% RSLogix 500 project LVD200607_TestA.RSS, saved by version 11.00.00.00 %
PROJECT "LINL0619"    % processor: type code 64 %

PROGRAM FILES
  LAD 2 "MAIN"  50 rungs  % Main Program Routine %
  LAD 4 "ENABLES"  14 rungs
  LAD 6 "FEED"  11 rungs  % normal %
  LAD 8 "SPEEDS"  12 rungs
  LAD 20 "HSC BOT"  5 rungs
  LAD 22 "HSC TOP"  5 rungs
  LAD 30 "1 MS STI"  17 rungs  % high speed %
  LAD 40 "SHIFT BOT"  8 rungs
  LAD 42 "SHIFT TOP"  16 rungs
  LAD 50 "BOTOPTIC"  3 rungs
  LAD 52 "BOTOPTMES"  7 rungs
  LAD 60 "1 INS1"  23 rungs
  LAD 61 "2 INS1RESU"  7 rungs
  LAD 62 "3 INS1PASS"  5 rungs
  LAD 63 "4 INS1FAIL"  3 rungs
  LAD 64 "5 INS1ACQ"  8 rungs
  LAD 65 "6 Q1TESTTR"  5 rungs
  LAD 66 "7 INS1TRIG"  5 rungs
  LAD 67 "8 FIFO1SET"  9 rungs
  LAD 68 "9 FIFO1GET"  8 rungs
  LAD 69 "10INSDATA1"  3 rungs
  LAD 70 "11TSTFALT1"  9 rungs
  LAD 71 "12INS1FIX1"  5 rungs
  LAD 72 "13INS1FIX2"  3 rungs
  LAD 73 "14 HSTRIG1"  5 rungs
  LAD 80 "XFER"  3 rungs
  LAD 90 "TOPOPTIC"  10 rungs
  LAD 91 "TOPOPVERT"  13 rungs
  LAD 92 "TOPOPREAL"  19 rungs
  LAD 93 "TOPOPTEST"  8 rungs
  LAD 94 "TOPOPRANGE"  6 rungs
  LAD 95 "TOPOPOKAY"  6 rungs
  LAD 96 "TESTINJECT"  8 rungs
  LAD 100 "1 INS5"  23 rungs
  LAD 101 "2 INS5RESU"  7 rungs
  LAD 102 "3 INS5PASS"  5 rungs
  LAD 103 "4 INS5FAIL"  3 rungs
  LAD 104 "5 INS5ACQ"  8 rungs
  LAD 105 "6 Q5TESTTR"  5 rungs
  LAD 106 "7 INS5TRIG"  5 rungs
  LAD 107 "8 FIFO5SET"  9 rungs
  LAD 108 "9 FIFO5GET"  8 rungs
  LAD 109 "10INSDATA5"  3 rungs
  LAD 110 "11TSTFALT5"  9 rungs
  LAD 111 "12INS5FIX1"  5 rungs
  LAD 112 "13INS5FIX2"  3 rungs
  LAD 113 "14 HSTRIG5"  5 rungs
  LAD 120 "1 INS6"  23 rungs
  LAD 121 "2 INS6RESU"  7 rungs
  LAD 122 "3 INS6PASS"  5 rungs
  LAD 123 "4 INS6FAIL"  3 rungs
  LAD 124 "5 INS6ACQ"  8 rungs
  LAD 125 "6 Q6TESTTR"  5 rungs
  LAD 126 "7 INS6TRIG"  5 rungs
  LAD 127 "8 FIFO6SET"  9 rungs
  LAD 128 "9 FIFO6GET"  8 rungs
  LAD 129 "10INSDATA6"  3 rungs
  LAD 130 "11TSTFALT6"  9 rungs
  LAD 131 "12INS6FIX1"  5 rungs
  LAD 132 "13INS6FIX2"  3 rungs
  LAD 133 "14 HSTRIG6"  5 rungs
  LAD 190 "PASS BLOW"  13 rungs
  LAD 201 "UNUSED"  14 rungs
  LAD 215 "TESTTRIG1"  4 rungs
  LAD 216 "TESTTRIG5"  4 rungs
  LAD 217 "TESTTRIG6"  4 rungs
  LAD 219 "PACKAGER"  28 rungs  % normal %
  LAD 220 "NO PACKAGE"  8 rungs
  LAD 222 "RATE1"  9 rungs
  LAD 223 "RATE2"  6 rungs
  LAD 224 "RESET RATE"  6 rungs
  LAD 240 "NP STOP"  8 rungs
  LAD 246 "SPEED BOT"  8 rungs  % high speed %
  LAD 248 "SPEED TOP"  8 rungs  % high speed %
  LAD 250 "P BOT"  7 rungs  % high speed %
  LAD 252 "P TOP"  7 rungs  % high speed %
  LAD 254 "TOTALCOUNT"  4 rungs
  LAD 255 "BLANK"  1 rungs
  LAD 74, 81, 114, 134, 191, 214, 218, 221, 225, 241: only END

DATA FILES
  O0 OUTPUT  11 elements
  I1 INPUT  11 elements
  S2 STATUS  66 elements
  B3 BINARY  14 elements
  T4 TIMER  45 elements
  C5 COUNTER  1 elements
  R6 CONTROL  30 elements
  N7 INTEGER  200 elements
  F8 FLOAT  100 elements
  B12 HMI_BINARY  22 elements  % general use with hmi to avoid additional reads %
  L13  COUNTS  256 elements
  F14 HMI_FLOATS  100 elements
  N15 HMI_INTS  100 elements
  L16 HMI_LONGS  100 elements
  L19 RATE DATA  50 elements
  L28 INS1TIME  50 elements
  L29 INS1POS  50 elements
  L30 INS5TIME  50 elements
  L31 INS5POS  50 elements
  L32 INS6TIME  50 elements
  L33 INS6POS  50 elements
  B34 BOT NG  128 elements
  B35 TOP NG  128 elements
  B36 BOTGOOD  128 elements
  B37 TOPGOOD  128 elements
  B38 EX1 TEST  128 elements
  B39 EX2GOOD  128 elements
  B40 EX2 TEST  128 elements
  N184 TEST INTS  50 elements
  L192 SPD OFFSET  50 elements
  B196 CTRL BITS  50 elements
  L199 USED  36 elements

LADDER 2 "MAIN"    % Main Program Routine %
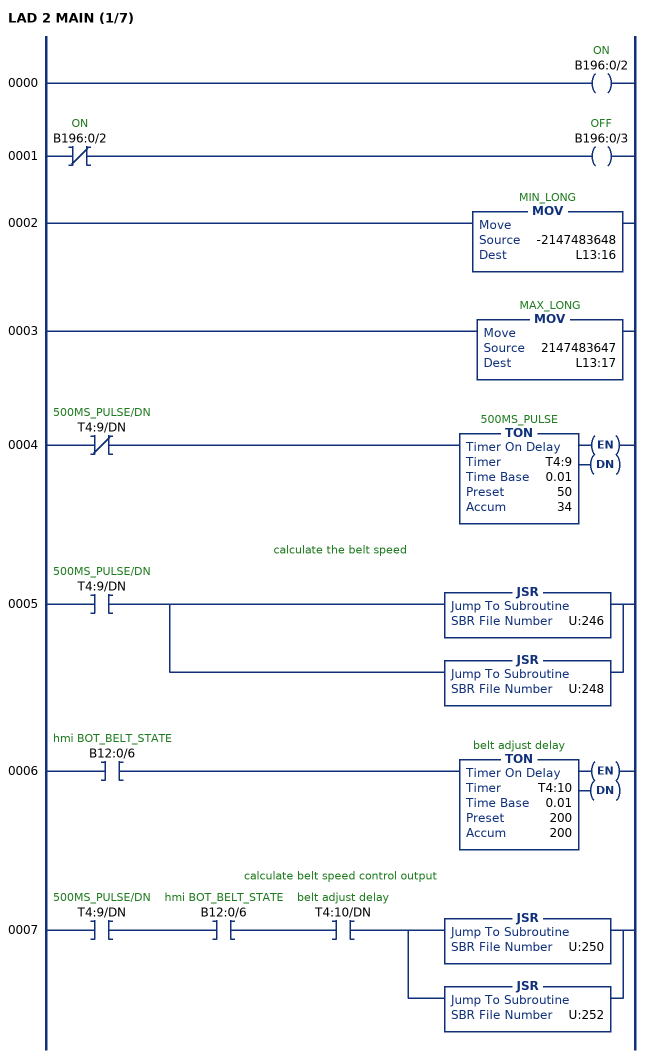
% Rung: 0 %
SOR OTE B196:0/2 EOR
%   B196:0/2  ON %
% Rung: 1 %
SOR XIO B196:0/2 OTE B196:0/3 EOR
%   B196:0/2  ON %
%   B196:0/3  OFF %
% Rung: 2 %
SOR MOV -2147483648 L13:16 EOR
%   L13:16  MIN_LONG %
% Rung: 3 %
SOR MOV 2147483647 L13:17 EOR
%   L13:17  MAX_LONG %
% Rung: 4 %
SOR XIO T4:9/DN TON T4:9 0.01 50 34 EOR
%   T4:9  500MS_PULSE %
% Rung: 5 %
% calculate the belt speed %
SOR XIC T4:9/DN BST JSR U:246 NXB JSR U:248 BND EOR
%   T4:9  500MS_PULSE %
% Rung: 6 %
SOR XIC B12:0/6 TON T4:10 0.01 200 200 EOR
%   B12:0/6  BOT_BELT_STATE  "hmi" %
%   T4:10  "belt adjust delay" %
% Rung: 7 %
% calculate belt speed control output %
SOR XIC T4:9/DN XIC B12:0/6 XIC T4:10/DN BST JSR U:250 NXB JSR U:252 BND EOR
%   T4:9  500MS_PULSE %
%   B12:0/6  BOT_BELT_STATE  "hmi" %
%   T4:10  "belt adjust delay" %

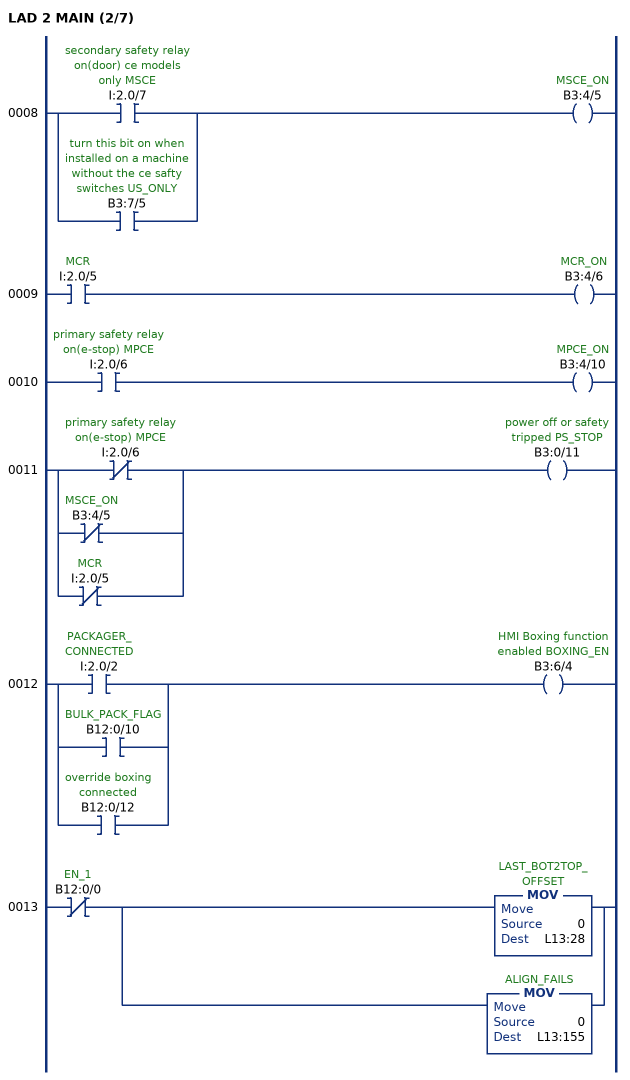
% Rung: 8 %
SOR BST XIC I:2.0/7 NXB XIC B3:7/5 BND OTE B3:4/5 EOR
%   I:2.0/7  MSCE  "secondary safety relay on(door) ce models only" %
%   B3:7/5  US_ONLY  "turn this bit on when installed on a machine without the ce safty switches" %
%   B3:4/5  MSCE_ON %
% Rung: 9 %
SOR XIC I:2.0/5 OTE B3:4/6 EOR
%   I:2.0/5  MCR %
%   B3:4/6  MCR_ON %
% Rung: 10 %
SOR XIC I:2.0/6 OTE B3:4/10 EOR
%   I:2.0/6  MPCE  "primary safety relay on(e-stop)" %
%   B3:4/10  MPCE_ON %
% Rung: 11 %
SOR BST XIO I:2.0/6 NXB XIO B3:4/5 NXB XIO I:2.0/5 BND OTE B3:0/11 EOR
%   I:2.0/6  MPCE  "primary safety relay on(e-stop)" %
%   B3:4/5  MSCE_ON %
%   I:2.0/5  MCR %
%   B3:0/11  PS_STOP  "power off or safety tripped" %
% Rung: 12 %
SOR BST XIC I:2.0/2 NXB XIC B12:0/10 NXB XIC B12:0/12 BND OTE B3:6/4 EOR
%   I:2.0/2  PACKAGER_CONNECTED %
%   B12:0/10  BULK_PACK_FLAG %
%   B12:0/12  "override boxing connected" %
%   B3:6/4  BOXING_EN  "HMI Boxing function enabled" %
% Rung: 13 %
SOR XIO B12:0/0 BST MOV 0 L13:28 NXB MOV 0 L13:155 BND EOR
%   B12:0/0  EN_1 %
%   L13:28  LAST_BOT2TOP_OFFSET %
%   L13:155  ALIGN_FAILS %

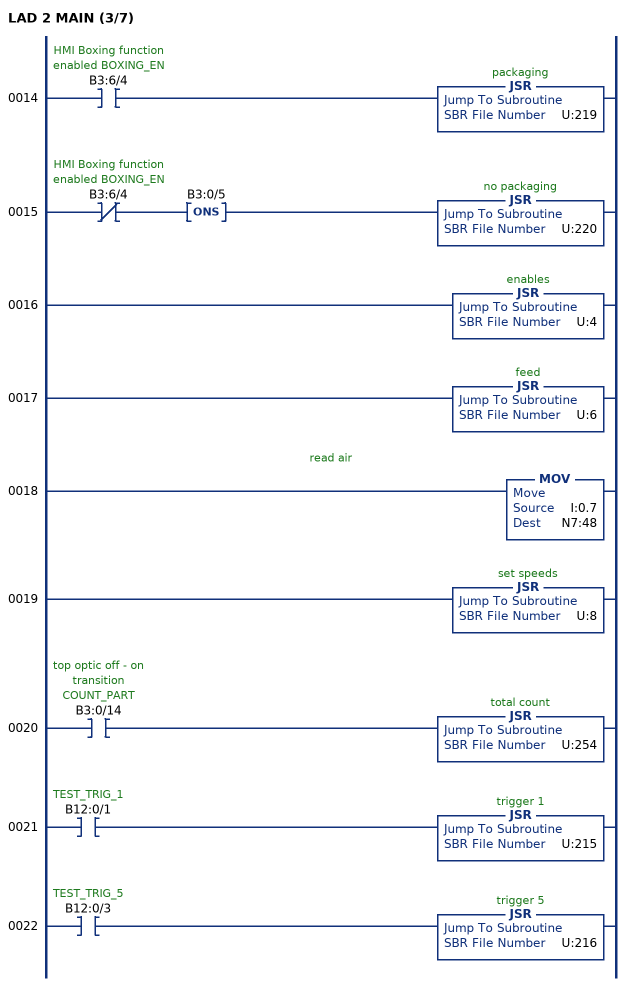
% Rung: 14 %
SOR XIC B3:6/4 JSR U:219 EOR
%   B3:6/4  BOXING_EN  "HMI Boxing function enabled" %
%   U:219  "packaging" %
% Rung: 15 %
SOR XIO B3:6/4 ONS B3:0/5 JSR U:220 EOR
%   B3:6/4  BOXING_EN  "HMI Boxing function enabled" %
%   U:220  "no packaging" %
% Rung: 16 %
SOR JSR U:4 EOR
%   U:4  "enables" %
% Rung: 17 %
SOR JSR U:6 EOR
%   U:6  "feed" %
% Rung: 18 %
% read air %
SOR MOV I:0.7 N7:48 EOR
%   I:0.7  "Air Presure Sensor Input Signal" %
% Rung: 19 %
SOR JSR U:8 EOR
%   U:8  "set speeds" %
% Rung: 20 %
SOR XIC B3:0/14 JSR U:254 EOR
%   B3:0/14  COUNT_PART  "top optic off - on transition" %
%   U:254  "total count" %
% Rung: 21 %
SOR XIC B12:0/1 JSR U:215 EOR
%   B12:0/1  TEST_TRIG_1 %
%   U:215  "trigger 1" %
% Rung: 22 %
SOR XIC B12:0/3 JSR U:216 EOR
%   B12:0/3  TEST_TRIG_5 %
%   U:216  "trigger 5" %

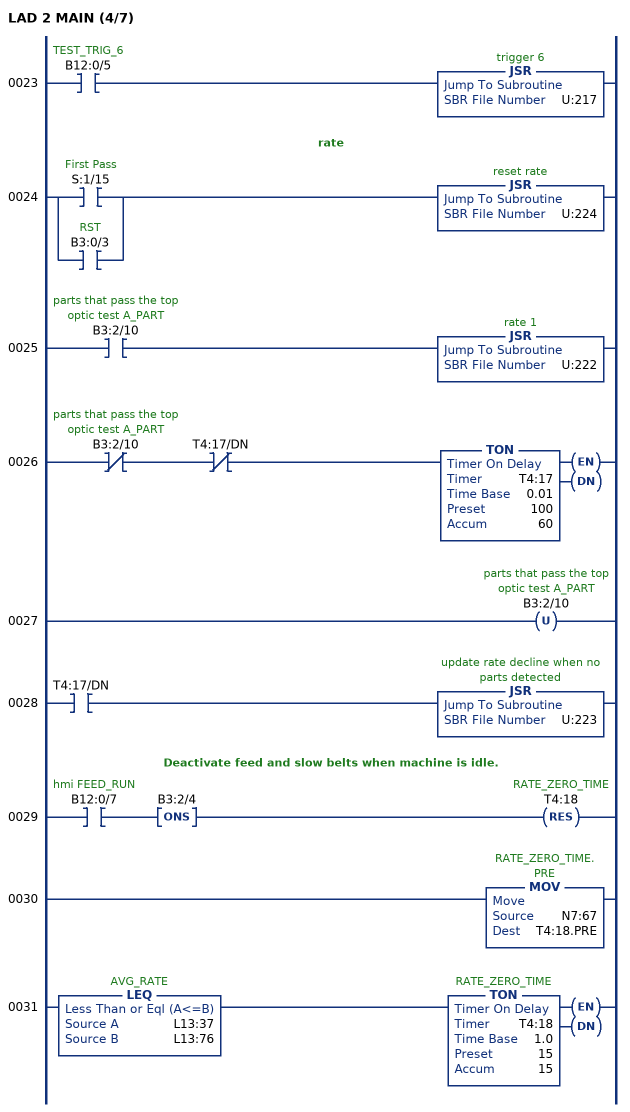
% Rung: 23 %
SOR XIC B12:0/5 JSR U:217 EOR
%   B12:0/5  TEST_TRIG_6 %
%   U:217  "trigger 6" %
% Rung: 24 %
% TITLE: rate %
SOR BST XIC S:1/15 NXB XIC B3:0/3 BND JSR U:224 EOR
%   S:1/15  "First Pass" %
%   B3:0/3  RST %
%   U:224  "reset rate" %
% Rung: 25 %
SOR XIC B3:2/10 JSR U:222 EOR
%   B3:2/10  A_PART  "parts that pass the top optic test" %
%   U:222  "rate 1" %
% Rung: 26 %
SOR XIO B3:2/10 XIO T4:17/DN TON T4:17 0.01 100 60 EOR
%   B3:2/10  A_PART  "parts that pass the top optic test" %
% Rung: 27 %
SOR OTU B3:2/10 EOR
%   B3:2/10  A_PART  "parts that pass the top optic test" %
% Rung: 28 %
SOR XIC T4:17/DN JSR U:223 EOR
%   U:223  "update rate decline when no parts detected" %
% Rung: 29 %
% TITLE: Deactivate feed and slow belts when machine is idle. %
SOR XIC B12:0/7 ONS B3:2/4 RES T4:18 EOR
%   B12:0/7  FEED_RUN  "hmi" %
%   T4:18  RATE_ZERO_TIME %
% Rung: 30 %
SOR MOV N7:67 T4:18.PRE EOR
%   N7:67  "empty bowl or jam bowl run time" %
%   T4:18  RATE_ZERO_TIME %
% Rung: 31 %
SOR LEQ L13:37 L13:76 TON T4:18 1.0 15 15 EOR
%   L13:37  AVG_RATE %
%   T4:18  RATE_ZERO_TIME %

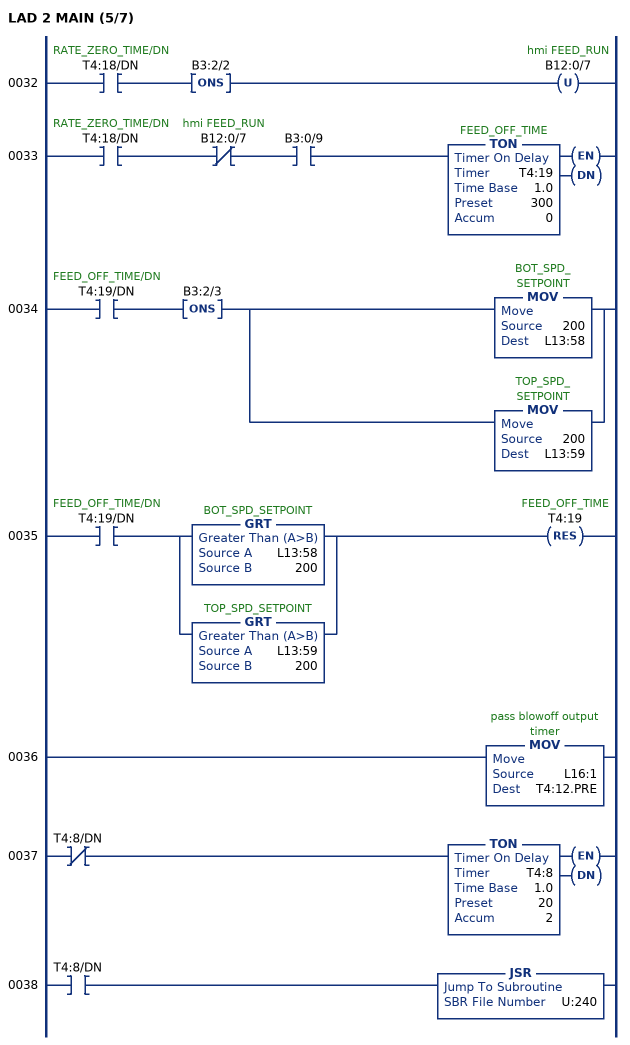
% Rung: 32 %
SOR XIC T4:18/DN ONS B3:2/2 OTU B12:0/7 EOR
%   T4:18  RATE_ZERO_TIME %
%   B12:0/7  FEED_RUN  "hmi" %
% Rung: 33 %
SOR XIC T4:18/DN XIO B12:0/7 XIC B3:0/9 TON T4:19 1.0 300 0 EOR
%   T4:18  RATE_ZERO_TIME %
%   B12:0/7  FEED_RUN  "hmi" %
%   T4:19  FEED_OFF_TIME %
% Rung: 34 %
SOR XIC T4:19/DN ONS B3:2/3 BST MOV 200 L13:58 NXB MOV 200 L13:59 BND EOR
%   T4:19  FEED_OFF_TIME %
%   L13:58  BOT_SPD_SETPOINT %
%   L13:59  TOP_SPD_SETPOINT %
% Rung: 35 %
SOR XIC T4:19/DN BST GRT L13:58 200 NXB GRT L13:59 200 BND RES T4:19 EOR
%   T4:19  FEED_OFF_TIME %
%   L13:58  BOT_SPD_SETPOINT %
%   L13:59  TOP_SPD_SETPOINT %
% Rung: 36 %
SOR MOV L16:1 T4:12.PRE EOR
%   L16:1  BLOW_TIME %
%   T4:12  "pass blowoff output timer" %
% Rung: 37 %
SOR XIO T4:8/DN TON T4:8 1.0 20 2 EOR
% Rung: 38 %
SOR XIC T4:8/DN JSR U:240 EOR

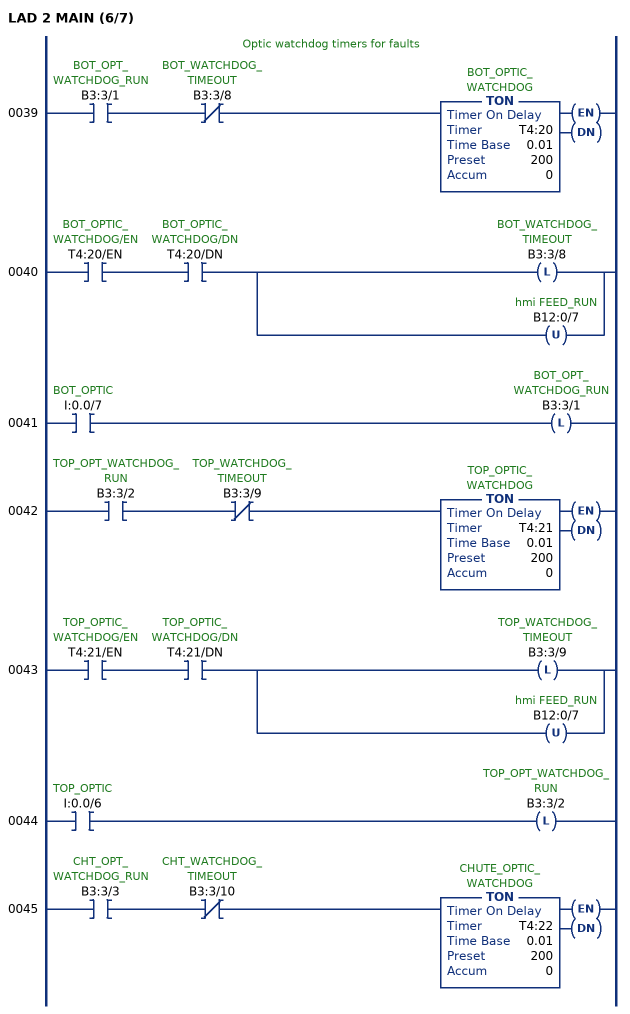
% Rung: 39 %
% Optic watchdog timers for faults %
SOR XIC B3:3/1 XIO B3:3/8 TON T4:20 0.01 200 0 EOR
%   B3:3/1  BOT_OPT_WATCHDOG_RUN %
%   B3:3/8  BOT_WATCHDOG_TIMEOUT %
%   T4:20  BOT_OPTIC_WATCHDOG %
% Rung: 40 %
SOR XIC T4:20/EN XIC T4:20/DN BST OTL B3:3/8 NXB OTU B12:0/7 BND EOR
%   T4:20  BOT_OPTIC_WATCHDOG %
%   B3:3/8  BOT_WATCHDOG_TIMEOUT %
%   B12:0/7  FEED_RUN  "hmi" %
% Rung: 41 %
SOR XIC I:0.0/7 OTL B3:3/1 EOR
%   I:0.0/7  BOT_OPTIC %
%   B3:3/1  BOT_OPT_WATCHDOG_RUN %
% Rung: 42 %
SOR XIC B3:3/2 XIO B3:3/9 TON T4:21 0.01 200 0 EOR
%   B3:3/2  TOP_OPT_WATCHDOG_RUN %
%   B3:3/9  TOP_WATCHDOG_TIMEOUT %
%   T4:21  TOP_OPTIC_WATCHDOG %
% Rung: 43 %
SOR XIC T4:21/EN XIC T4:21/DN BST OTL B3:3/9 NXB OTU B12:0/7 BND EOR
%   T4:21  TOP_OPTIC_WATCHDOG %
%   B3:3/9  TOP_WATCHDOG_TIMEOUT %
%   B12:0/7  FEED_RUN  "hmi" %
% Rung: 44 %
SOR XIC I:0.0/6 OTL B3:3/2 EOR
%   I:0.0/6  TOP_OPTIC %
%   B3:3/2  TOP_OPT_WATCHDOG_RUN %
% Rung: 45 %
SOR XIC B3:3/3 XIO B3:3/10 TON T4:22 0.01 200 0 EOR
%   B3:3/3  CHT_OPT_WATCHDOG_RUN %
%   B3:3/10  CHT_WATCHDOG_TIMEOUT %
%   T4:22  CHUTE_OPTIC_WATCHDOG %

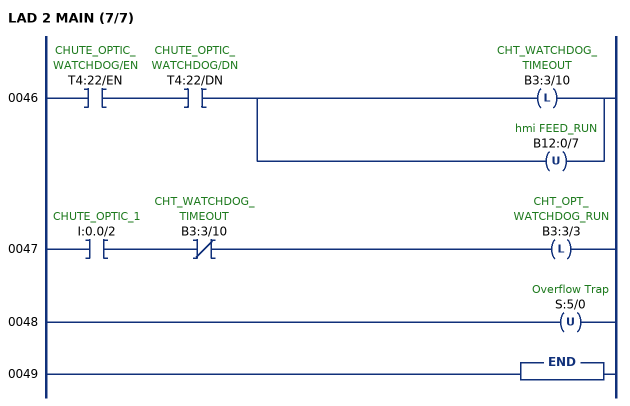
% Rung: 46 %
SOR XIC T4:22/EN XIC T4:22/DN BST OTL B3:3/10 NXB OTU B12:0/7 BND EOR
%   T4:22  CHUTE_OPTIC_WATCHDOG %
%   B3:3/10  CHT_WATCHDOG_TIMEOUT %
%   B12:0/7  FEED_RUN  "hmi" %
% Rung: 47 %
SOR XIC I:0.0/2 XIO B3:3/10 OTL B3:3/3 EOR
%   I:0.0/2  CHUTE_OPTIC_1 %
%   B3:3/10  CHT_WATCHDOG_TIMEOUT %
%   B3:3/3  CHT_OPT_WATCHDOG_RUN %
% Rung: 48 %
SOR OTU S:5/0 EOR
%   S:5/0  "Overflow Trap" %
% Rung: 49 %
SOR END EOR

LADDER 4 "ENABLES"
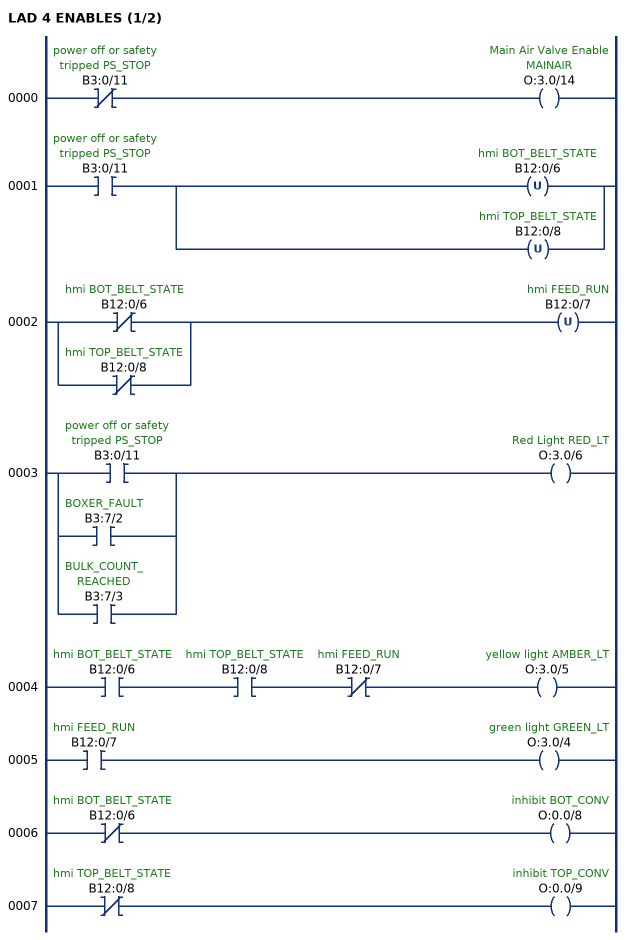
% Rung: 0 %
SOR XIO B3:0/11 OTE O:3.0/14 EOR
%   B3:0/11  PS_STOP  "power off or safety tripped" %
%   O:3.0/14  MAINAIR  "Main Air Valve Enable" %
% Rung: 1 %
SOR XIC B3:0/11 BST OTU B12:0/6 NXB OTU B12:0/8 BND EOR
%   B3:0/11  PS_STOP  "power off or safety tripped" %
%   B12:0/6  BOT_BELT_STATE  "hmi" %
%   B12:0/8  TOP_BELT_STATE  "hmi" %
% Rung: 2 %
SOR BST XIO B12:0/6 NXB XIO B12:0/8 BND OTU B12:0/7 EOR
%   B12:0/6  BOT_BELT_STATE  "hmi" %
%   B12:0/8  TOP_BELT_STATE  "hmi" %
%   B12:0/7  FEED_RUN  "hmi" %
% Rung: 3 %
SOR BST XIC B3:0/11 NXB XIC B3:7/2 NXB XIC B3:7/3 BND OTE O:3.0/6 EOR
%   B3:0/11  PS_STOP  "power off or safety tripped" %
%   B3:7/2  BOXER_FAULT %
%   B3:7/3  BULK_COUNT_REACHED %
%   O:3.0/6  RED_LT  "Red Light" %
% Rung: 4 %
SOR XIC B12:0/6 XIC B12:0/8 XIO B12:0/7 OTE O:3.0/5 EOR
%   B12:0/6  BOT_BELT_STATE  "hmi" %
%   B12:0/8  TOP_BELT_STATE  "hmi" %
%   B12:0/7  FEED_RUN  "hmi" %
%   O:3.0/5  AMBER_LT  "yellow light" %
% Rung: 5 %
SOR XIC B12:0/7 OTE O:3.0/4 EOR
%   B12:0/7  FEED_RUN  "hmi" %
%   O:3.0/4  GREEN_LT  "green light" %
% Rung: 6 %
SOR XIO B12:0/6 OTE O:0.0/8 EOR
%   B12:0/6  BOT_BELT_STATE  "hmi" %
%   O:0.0/8  BOT_CONV  "inhibit" %
% Rung: 7 %
SOR XIO B12:0/8 OTE O:0.0/9 EOR
%   B12:0/8  TOP_BELT_STATE  "hmi" %
%   O:0.0/9  TOP_CONV  "inhibit" %

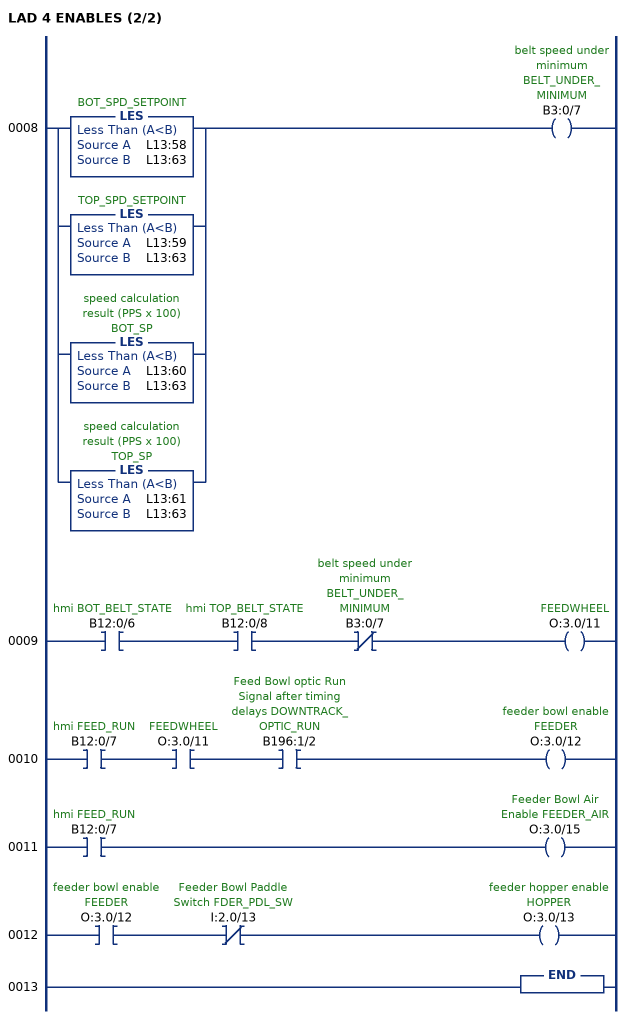
% Rung: 8 %
SOR BST LES L13:58 L13:63 NXB LES L13:59 L13:63 NXB LES L13:60 L13:63 NXB LES L13:61 L13:63 BND OTE B3:0/7 EOR
%   L13:58  BOT_SPD_SETPOINT %
%   L13:63  "min belt speed" %
%   L13:59  TOP_SPD_SETPOINT %
%   L13:60  BOT_SP  "speed calculation result (PPS x 100)" %
%   L13:61  TOP_SP  "speed calculation result (PPS x 100)" %
%   B3:0/7  BELT_UNDER_MINIMUM  "belt speed under minimum" %
% Rung: 9 %
SOR XIC B12:0/6 XIC B12:0/8 XIO B3:0/7 OTE O:3.0/11 EOR
%   B12:0/6  BOT_BELT_STATE  "hmi" %
%   B12:0/8  TOP_BELT_STATE  "hmi" %
%   B3:0/7  BELT_UNDER_MINIMUM  "belt speed under minimum" %
%   O:3.0/11  FEEDWHEEL %
% Rung: 10 %
SOR XIC B12:0/7 XIC O:3.0/11 XIC B196:1/2 OTE O:3.0/12 EOR
%   B12:0/7  FEED_RUN  "hmi" %
%   O:3.0/11  FEEDWHEEL %
%   B196:1/2  DOWNTRACK_OPTIC_RUN  "Feed Bowl optic Run Signal after timing delays" %
%   O:3.0/12  FEEDER  "feeder bowl enable" %
% Rung: 11 %
SOR XIC B12:0/7 OTE O:3.0/15 EOR
%   B12:0/7  FEED_RUN  "hmi" %
%   O:3.0/15  FEEDER_AIR  "Feeder Bowl Air Enable" %
% Rung: 12 %
SOR XIC O:3.0/12 XIO I:2.0/13 OTE O:3.0/13 EOR
%   O:3.0/12  FEEDER  "feeder bowl enable" %
%   I:2.0/13  FDER_PDL_SW  "Feeder Bowl Paddle Switch" %
%   O:3.0/13  HOPPER  "feeder hopper enable" %
% Rung: 13 %
SOR END EOR

LADDER 6 "FEED"    % normal %
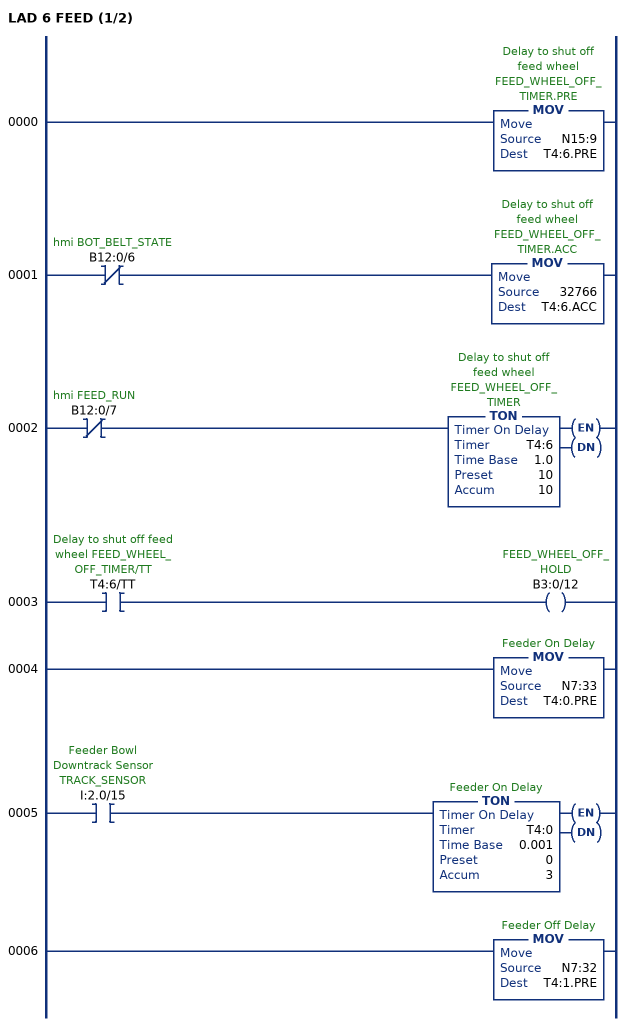
% Rung: 0 %
SOR MOV N15:9 T4:6.PRE EOR
%   N15:9  FEED_WHEEL_STOP_TIME %
%   T4:6  FEED_WHEEL_OFF_TIMER  "Delay to shut off feed wheel" %
% Rung: 1 %
SOR XIO B12:0/6 MOV 32766 T4:6.ACC EOR
%   B12:0/6  BOT_BELT_STATE  "hmi" %
%   T4:6  FEED_WHEEL_OFF_TIMER  "Delay to shut off feed wheel" %
% Rung: 2 %
SOR XIO B12:0/7 TON T4:6 1.0 10 10 EOR
%   B12:0/7  FEED_RUN  "hmi" %
%   T4:6  FEED_WHEEL_OFF_TIMER  "Delay to shut off feed wheel" %
% Rung: 3 %
SOR XIC T4:6/TT OTE B3:0/12 EOR
%   T4:6  FEED_WHEEL_OFF_TIMER  "Delay to shut off feed wheel" %
%   B3:0/12  FEED_WHEEL_OFF_HOLD %
% Rung: 4 %
SOR MOV N7:33 T4:0.PRE EOR
%   N7:33  "down track on delay" %
%   T4:0  "Feeder On Delay" %
% Rung: 5 %
SOR XIC I:2.0/15 TON T4:0 0.001 0 3 EOR
%   I:2.0/15  TRACK_SENSOR  "Feeder Bowl Downtrack Sensor" %
%   T4:0  "Feeder On Delay" %
% Rung: 6 %
SOR MOV N7:32 T4:1.PRE EOR
%   N7:32  "down track off delay" %
%   T4:1  "Feeder Off Delay" %

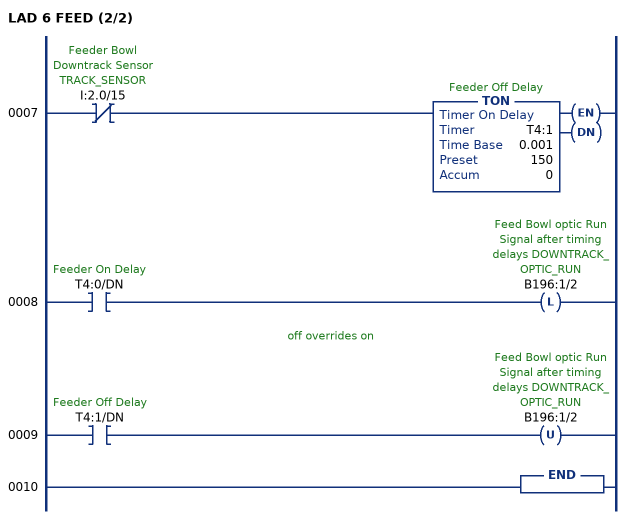
% Rung: 7 %
SOR XIO I:2.0/15 TON T4:1 0.001 150 0 EOR
%   I:2.0/15  TRACK_SENSOR  "Feeder Bowl Downtrack Sensor" %
%   T4:1  "Feeder Off Delay" %
% Rung: 8 %
SOR XIC T4:0/DN OTL B196:1/2 EOR
%   T4:0  "Feeder On Delay" %
%   B196:1/2  DOWNTRACK_OPTIC_RUN  "Feed Bowl optic Run Signal after timing delays" %
% Rung: 9 %
% off overrides on %
SOR XIC T4:1/DN OTU B196:1/2 EOR
%   T4:1  "Feeder Off Delay" %
%   B196:1/2  DOWNTRACK_OPTIC_RUN  "Feed Bowl optic Run Signal after timing delays" %
% Rung: 10 %
SOR END EOR

LADDER 8 "SPEEDS"
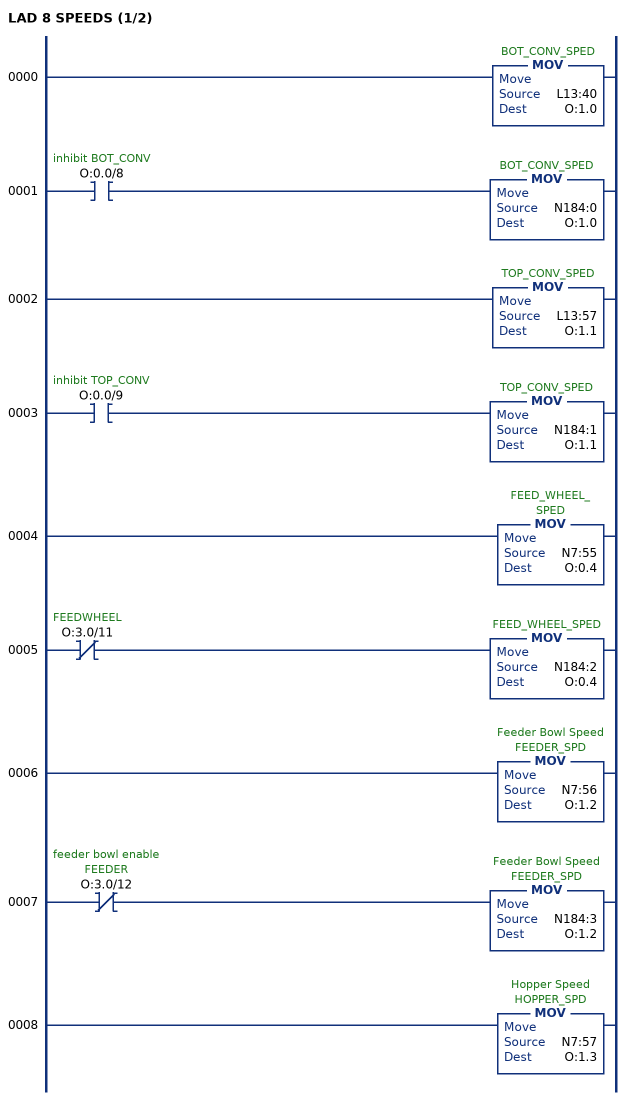
% Rung: 0 %
SOR MOV L13:40 O:1.0 EOR
%   L13:40  SCALED_BOT_VALUE %
%   O:1.0  BOT_CONV_SPED %
% Rung: 1 %
SOR XIC O:0.0/8 MOV N184:0 O:1.0 EOR
%   O:0.0/8  BOT_CONV  "inhibit" %
%   O:1.0  BOT_CONV_SPED %
% Rung: 2 %
SOR MOV L13:57 O:1.1 EOR
%   L13:57  SCALED_TOP_VALUE %
%   O:1.1  TOP_CONV_SPED %
% Rung: 3 %
SOR XIC O:0.0/9 MOV N184:1 O:1.1 EOR
%   O:0.0/9  TOP_CONV  "inhibit" %
%   O:1.1  TOP_CONV_SPED %
% Rung: 4 %
SOR MOV N7:55 O:0.4 EOR
%   O:0.4  FEED_WHEEL_SPED %
% Rung: 5 %
SOR XIO O:3.0/11 MOV N184:2 O:0.4 EOR
%   O:3.0/11  FEEDWHEEL %
%   O:0.4  FEED_WHEEL_SPED %
% Rung: 6 %
SOR MOV N7:56 O:1.2 EOR
%   O:1.2  FEEDER_SPD  "Feeder Bowl Speed" %
% Rung: 7 %
SOR XIO O:3.0/12 MOV N184:3 O:1.2 EOR
%   O:3.0/12  FEEDER  "feeder bowl enable" %
%   O:1.2  FEEDER_SPD  "Feeder Bowl Speed" %
% Rung: 8 %
SOR MOV N7:57 O:1.3 EOR
%   O:1.3  HOPPER_SPD  "Hopper Speed" %

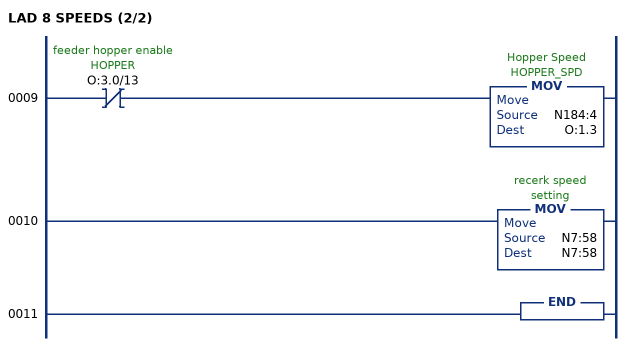
% Rung: 9 %
SOR XIO O:3.0/13 MOV N184:4 O:1.3 EOR
%   O:3.0/13  HOPPER  "feeder hopper enable" %
%   O:1.3  HOPPER_SPD  "Hopper Speed" %
% Rung: 10 %
SOR MOV N7:58 N7:58 EOR
%   N7:58  "recerk speed setting" %
% Rung: 11 %
SOR END EOR

LADDER 20 "HSC BOT"
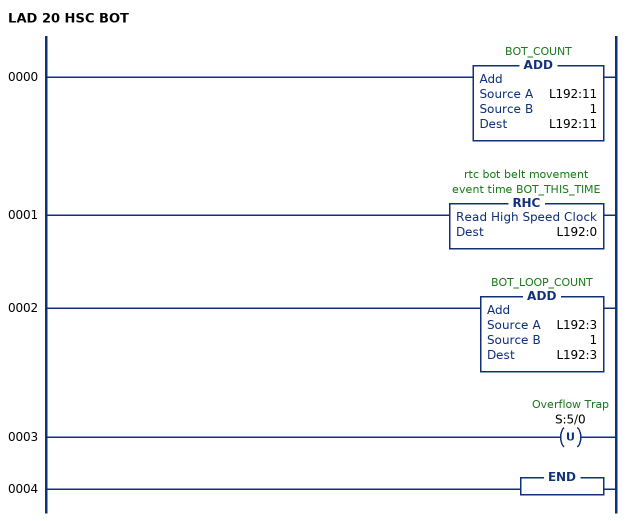
% Rung: 0 %
SOR ADD L192:11 1 L192:11 EOR
%   L192:11  BOT_COUNT %
% Rung: 1 %
SOR RHC L192:0 EOR
%   L192:0  BOT_THIS_TIME  "rtc bot belt movement event time" %
% Rung: 2 %
SOR ADD L192:3 1 L192:3 EOR
%   L192:3  BOT_LOOP_COUNT %
% Rung: 3 %
SOR OTU S:5/0 EOR
%   S:5/0  "Overflow Trap" %
% Rung: 4 %
SOR END EOR

LADDER 22 "HSC TOP"
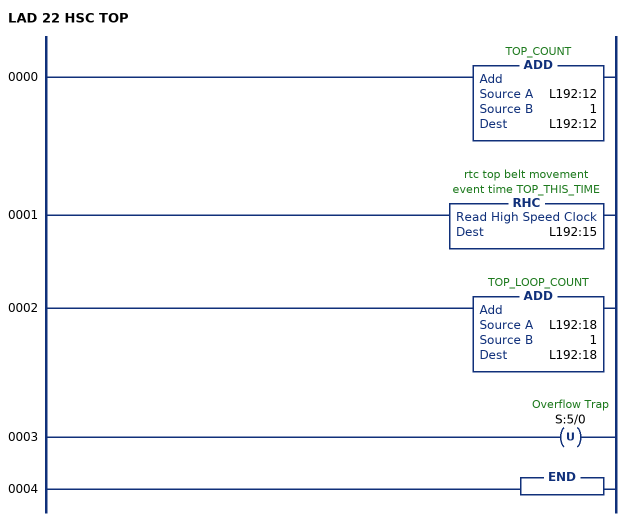
% Rung: 0 %
SOR ADD L192:12 1 L192:12 EOR
%   L192:12  TOP_COUNT %
% Rung: 1 %
SOR RHC L192:15 EOR
%   L192:15  TOP_THIS_TIME  "rtc top belt movement event time" %
% Rung: 2 %
SOR ADD L192:18 1 L192:18 EOR
%   L192:18  TOP_LOOP_COUNT %
% Rung: 3 %
SOR OTU S:5/0 EOR
%   S:5/0  "Overflow Trap" %
% Rung: 4 %
SOR END EOR

LADDER 30 "1 MS STI"    % high speed %
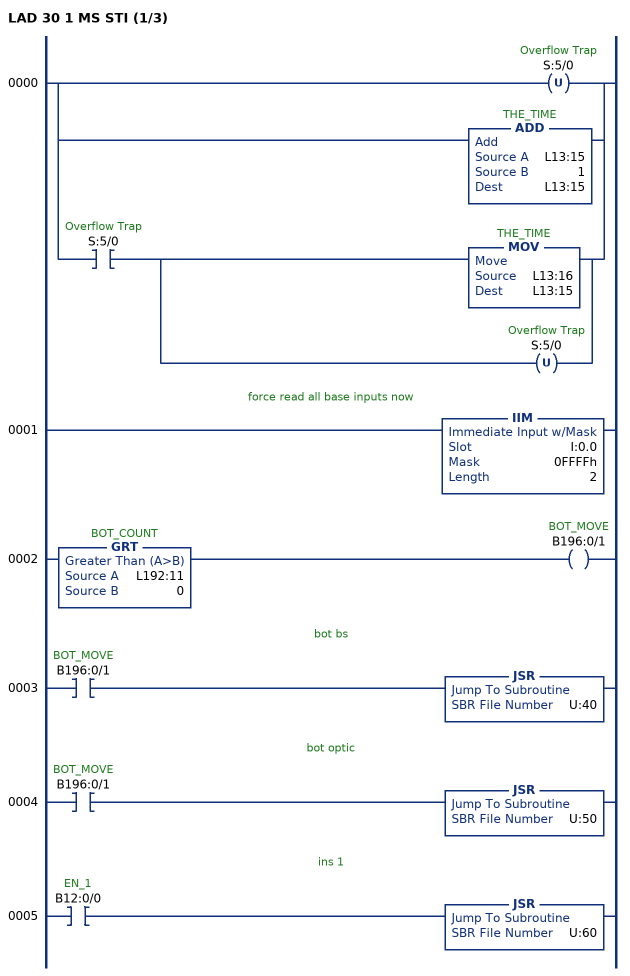
% Rung: 0 %
SOR BST OTU S:5/0 NXB ADD L13:15 1 L13:15 NXB XIC S:5/0 BST MOV L13:16 L13:15 NXB OTU S:5/0 BND BND EOR
%   S:5/0  "Overflow Trap" %
%   L13:15  THE_TIME %
%   L13:16  MIN_LONG %
% Rung: 1 %
% force read all base inputs now %
SOR IIM I:0.0 0FFFFh 2 EOR
% Rung: 2 %
SOR GRT L192:11 0 OTE B196:0/1 EOR
%   L192:11  BOT_COUNT %
%   B196:0/1  BOT_MOVE %
% Rung: 3 %
% bot bs %
SOR XIC B196:0/1 JSR U:40 EOR
%   B196:0/1  BOT_MOVE %
% Rung: 4 %
% bot optic %
SOR XIC B196:0/1 JSR U:50 EOR
%   B196:0/1  BOT_MOVE %
% Rung: 5 %
% ins 1 %
SOR XIC B12:0/0 JSR U:60 EOR
%   B12:0/0  EN_1 %

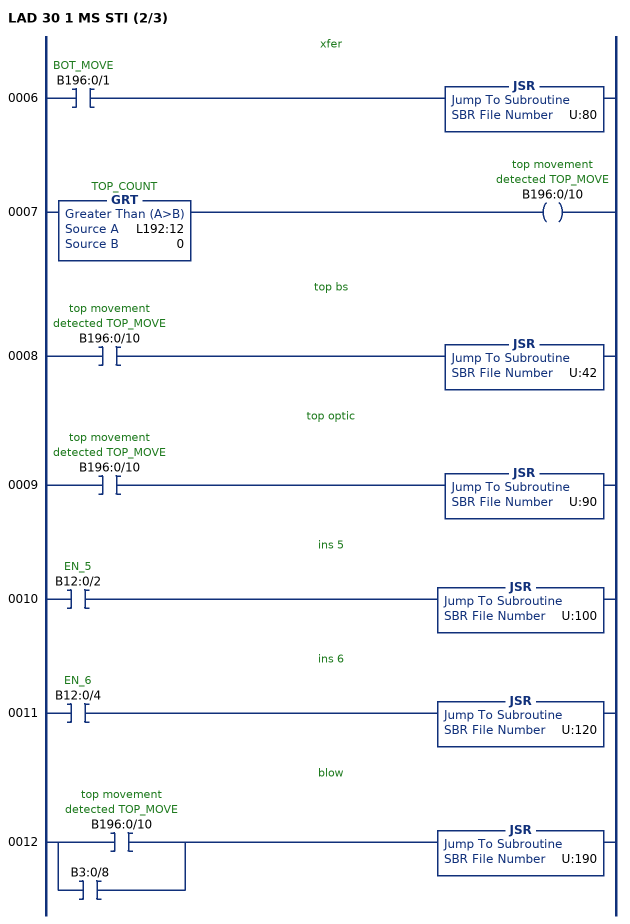
% Rung: 6 %
% xfer %
SOR XIC B196:0/1 JSR U:80 EOR
%   B196:0/1  BOT_MOVE %
% Rung: 7 %
SOR GRT L192:12 0 OTE B196:0/10 EOR
%   L192:12  TOP_COUNT %
%   B196:0/10  TOP_MOVE  "top movement detected" %
% Rung: 8 %
% top bs %
SOR XIC B196:0/10 JSR U:42 EOR
%   B196:0/10  TOP_MOVE  "top movement detected" %
% Rung: 9 %
% top optic %
SOR XIC B196:0/10 JSR U:90 EOR
%   B196:0/10  TOP_MOVE  "top movement detected" %
% Rung: 10 %
% ins 5 %
SOR XIC B12:0/2 JSR U:100 EOR
%   B12:0/2  EN_5 %
% Rung: 11 %
% ins 6 %
SOR XIC B12:0/4 JSR U:120 EOR
%   B12:0/4  EN_6 %
% Rung: 12 %
% blow %
SOR BST XIC B196:0/10 NXB XIC B3:0/8 BND JSR U:190 EOR
%   B196:0/10  TOP_MOVE  "top movement detected" %

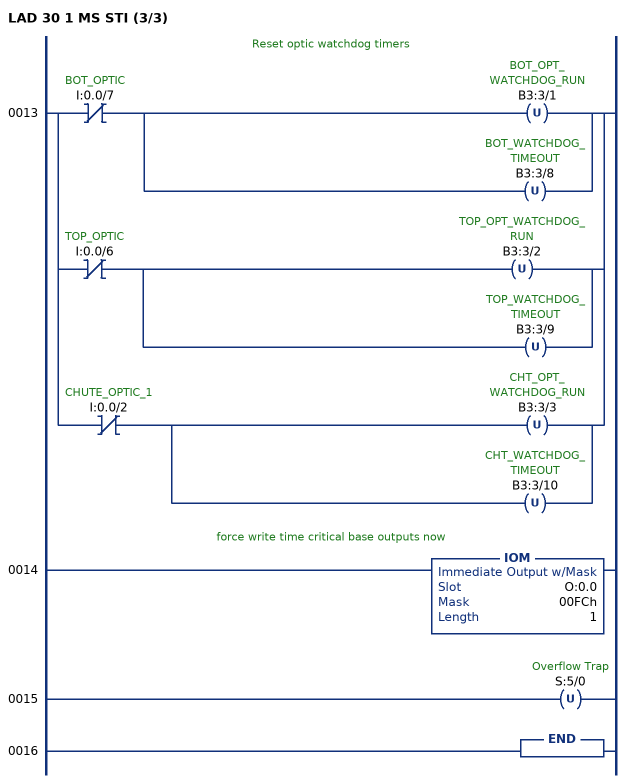
% Rung: 13 %
% Reset optic watchdog timers %
SOR BST XIO I:0.0/7 BST OTU B3:3/1 NXB OTU B3:3/8 BND NXB XIO I:0.0/6 BST OTU B3:3/2 NXB OTU B3:3/9 BND NXB XIO I:0.0/2 BST OTU B3:3/3 NXB OTU B3:3/10 BND BND EOR
%   I:0.0/7  BOT_OPTIC %
%   B3:3/1  BOT_OPT_WATCHDOG_RUN %
%   B3:3/8  BOT_WATCHDOG_TIMEOUT %
%   I:0.0/6  TOP_OPTIC %
%   B3:3/2  TOP_OPT_WATCHDOG_RUN %
%   B3:3/9  TOP_WATCHDOG_TIMEOUT %
%   I:0.0/2  CHUTE_OPTIC_1 %
%   B3:3/3  CHT_OPT_WATCHDOG_RUN %
%   B3:3/10  CHT_WATCHDOG_TIMEOUT %
% Rung: 14 %
% force write time critical base outputs now %
SOR IOM O:0.0 00FCh 1 EOR
% Rung: 15 %
SOR OTU S:5/0 EOR
%   S:5/0  "Overflow Trap" %
% Rung: 16 %
SOR END EOR

LADDER 40 "SHIFT BOT"
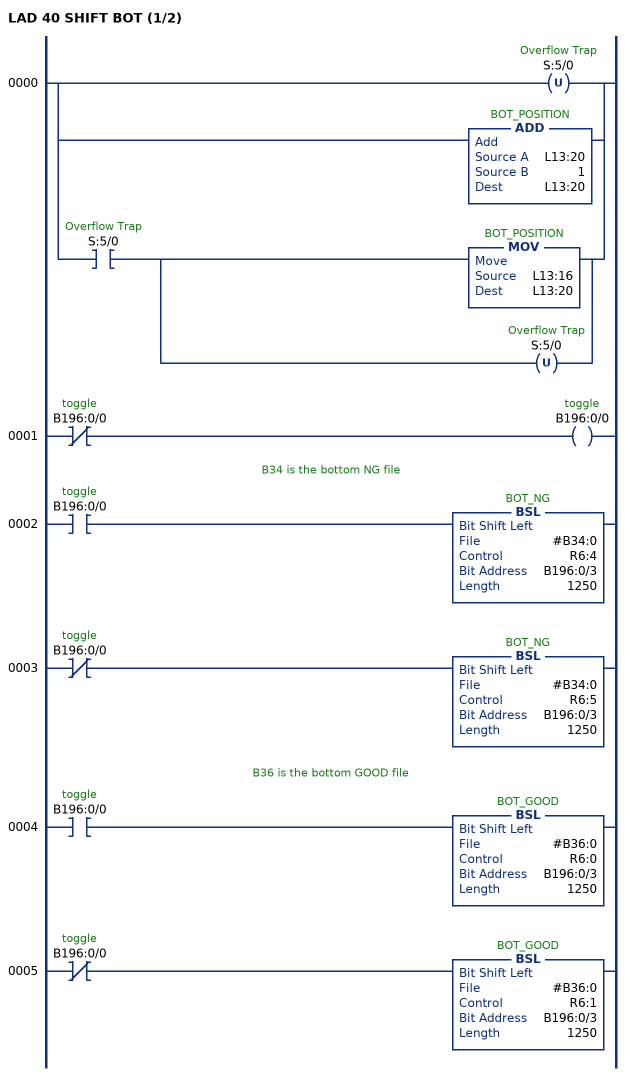
% Rung: 0 %
SOR BST OTU S:5/0 NXB ADD L13:20 1 L13:20 NXB XIC S:5/0 BST MOV L13:16 L13:20 NXB OTU S:5/0 BND BND EOR
%   S:5/0  "Overflow Trap" %
%   L13:20  BOT_POSITION %
%   L13:16  MIN_LONG %
% Rung: 1 %
SOR XIO B196:0/0 OTE B196:0/0 EOR
%   B196:0/0  "toggle" %
% Rung: 2 %
% B34 is the bottom NG file %
SOR XIC B196:0/0 BSL #B34:0 R6:4 B196:0/3 1250 EOR
%   B196:0/0  "toggle" %
%   B34:0  BOT_NG %
%   B196:0/3  OFF %
% Rung: 3 %
SOR XIO B196:0/0 BSL #B34:0 R6:5 B196:0/3 1250 EOR
%   B196:0/0  "toggle" %
%   B34:0  BOT_NG %
%   B196:0/3  OFF %
% Rung: 4 %
% B36 is the bottom GOOD file %
SOR XIC B196:0/0 BSL #B36:0 R6:0 B196:0/3 1250 EOR
%   B196:0/0  "toggle" %
%   B36:0  BOT_GOOD %
%   B196:0/3  OFF %
% Rung: 5 %
SOR XIO B196:0/0 BSL #B36:0 R6:1 B196:0/3 1250 EOR
%   B196:0/0  "toggle" %
%   B36:0  BOT_GOOD %
%   B196:0/3  OFF %

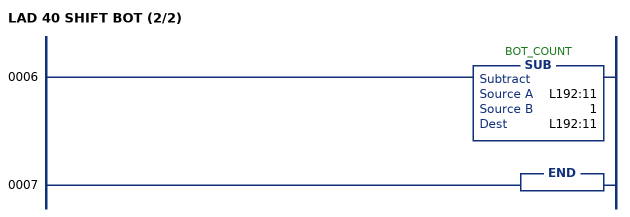
% Rung: 6 %
SOR SUB L192:11 1 L192:11 EOR
%   L192:11  BOT_COUNT %
% Rung: 7 %
SOR END EOR

LADDER 42 "SHIFT TOP"
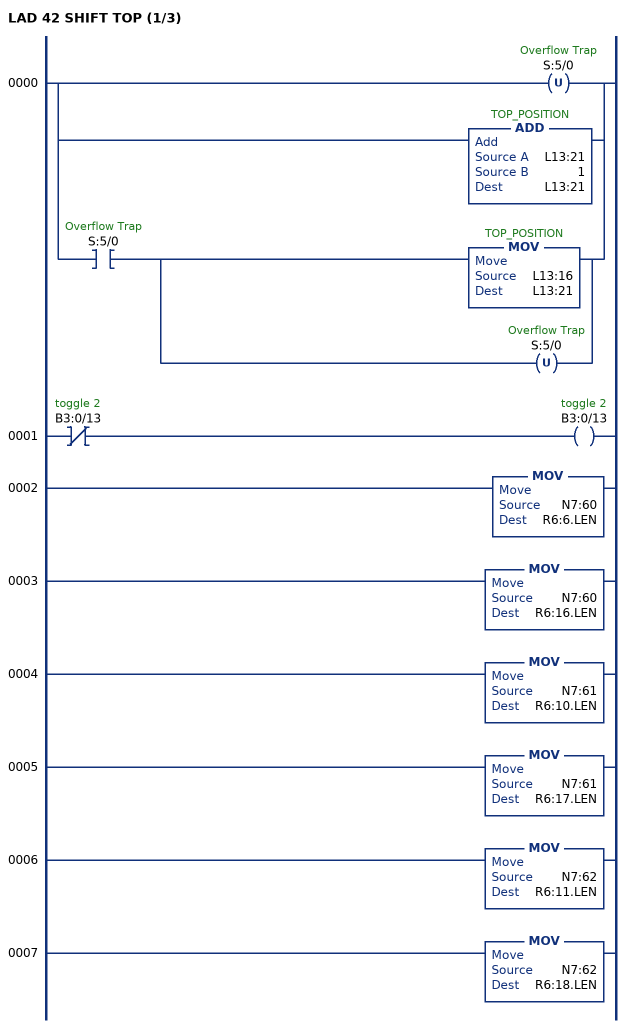
% Rung: 0 %
SOR BST OTU S:5/0 NXB ADD L13:21 1 L13:21 NXB XIC S:5/0 BST MOV L13:16 L13:21 NXB OTU S:5/0 BND BND EOR
%   S:5/0  "Overflow Trap" %
%   L13:21  TOP_POSITION %
%   L13:16  MIN_LONG %
% Rung: 1 %
SOR XIO B3:0/13 OTE B3:0/13 EOR
%   B3:0/13  "toggle 2" %
% Rung: 2 %
SOR MOV N7:60 R6:6.LEN EOR
% Rung: 3 %
SOR MOV N7:60 R6:16.LEN EOR
% Rung: 4 %
SOR MOV N7:61 R6:10.LEN EOR
% Rung: 5 %
SOR MOV N7:61 R6:17.LEN EOR
% Rung: 6 %
SOR MOV N7:62 R6:11.LEN EOR
% Rung: 7 %
SOR MOV N7:62 R6:18.LEN EOR

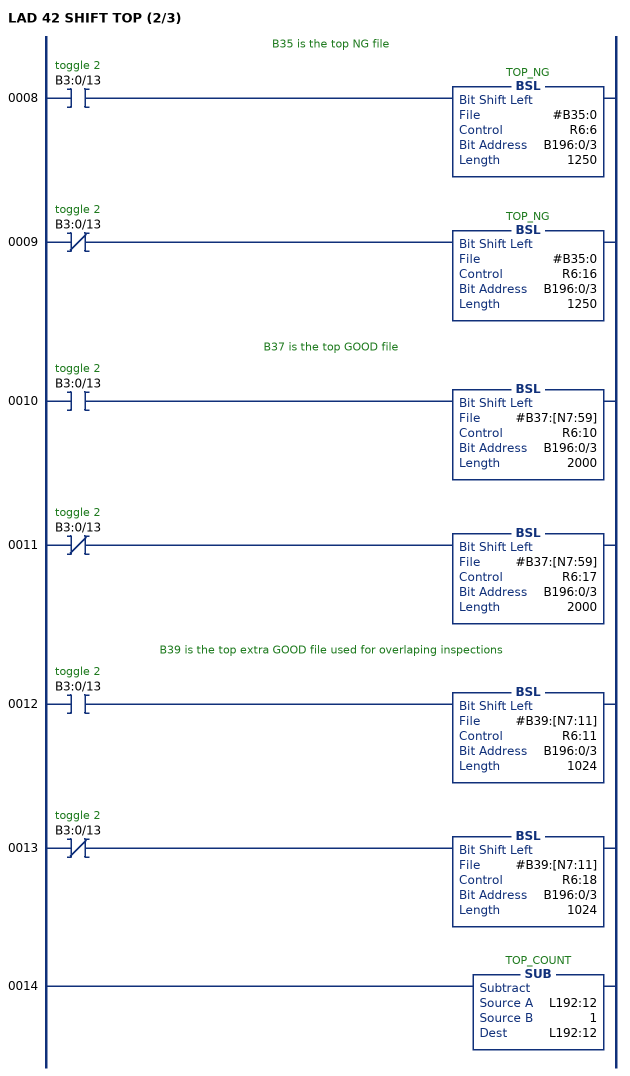
% Rung: 8 %
% B35 is the top NG file %
SOR XIC B3:0/13 BSL #B35:0 R6:6 B196:0/3 1250 EOR
%   B3:0/13  "toggle 2" %
%   B35:0  TOP_NG %
%   B196:0/3  OFF %
% Rung: 9 %
SOR XIO B3:0/13 BSL #B35:0 R6:16 B196:0/3 1250 EOR
%   B3:0/13  "toggle 2" %
%   B35:0  TOP_NG %
%   B196:0/3  OFF %
% Rung: 10 %
% B37 is the top GOOD file %
SOR XIC B3:0/13 BSL #B37:[N7:59] R6:10 B196:0/3 2000 EOR
%   B3:0/13  "toggle 2" %
%   B196:0/3  OFF %
% Rung: 11 %
SOR XIO B3:0/13 BSL #B37:[N7:59] R6:17 B196:0/3 2000 EOR
%   B3:0/13  "toggle 2" %
%   B196:0/3  OFF %
% Rung: 12 %
% B39 is the top extra GOOD file used for overlaping inspections %
SOR XIC B3:0/13 BSL #B39:[N7:11] R6:11 B196:0/3 1024 EOR
%   B3:0/13  "toggle 2" %
%   B196:0/3  OFF %
% Rung: 13 %
SOR XIO B3:0/13 BSL #B39:[N7:11] R6:18 B196:0/3 1024 EOR
%   B3:0/13  "toggle 2" %
%   B196:0/3  OFF %
% Rung: 14 %
SOR SUB L192:12 1 L192:12 EOR
%   L192:12  TOP_COUNT %

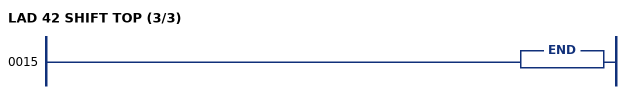
% Rung: 15 %
SOR END EOR

LADDER 50 "BOTOPTIC"
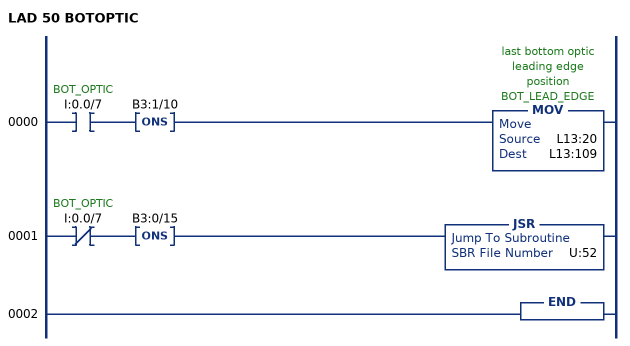
% Rung: 0 %
SOR XIC I:0.0/7 ONS B3:1/10 MOV L13:20 L13:109 EOR
%   I:0.0/7  BOT_OPTIC %
%   L13:20  BOT_POSITION %
%   L13:109  BOT_LEAD_EDGE  "last bottom optic leading edge position" %
% Rung: 1 %
SOR XIO I:0.0/7 ONS B3:0/15 JSR U:52 EOR
%   I:0.0/7  BOT_OPTIC %
% Rung: 2 %
SOR END EOR

LADDER 52 "BOTOPTMES"
